PROGRAM MAIN
VAR
	fbGetCurTaskIdx  : GETCURTASKINDEX;
	
	Layout : Buffer_Layout;
	Buffer : ARRAY[0..63] OF BYTE;
	
	// out var
	VarEen : INT;
	VarTwee : INT;
END_VAR


Set_Buffer_Layout(
	Buffer_Size:= 64, 
	Bool_Amount:= 0, 
	Int_Amount:= 0, 
	Real_Amount:= 0, 
	String_Amount:= 2, 
	Layout:= Layout);

Set_Int_From_Buffer(
	In:= 300, 
	Num:= 0, 
	Layout:= Layout, 
	Buffer:= Buffer);
	
Set_Int_From_Buffer(
	In:= 30, 
	Num:= 1, 
	Layout:= Layout, 
	Buffer:= Buffer);
	
Set_Bool_Fom_Buffer(
	In:= TRUE, 
	Num:= 0, 
	Layout:= Layout, 
	Buffer:= Buffer);
	
	
Set_Bool_Fom_Buffer(
	In:= TRUE, 
	Num:= 1, 
	Layout:= Layout, 
	Buffer:= Buffer);
	
	
Set_Real_From_Buffer(
	In:= 3.55, 
	Num:= 0, 
	Layout:= Layout, 
	Buffer:= Buffer);
	
Set_Real_From_Buffer(
	In:= 10.66, 
	Num:= 1, 
	Layout:= Layout, 
	Buffer:= Buffer);
	
	
Set_String_From_Buffer(
	In:= 'AAAAA', 
	Num:= 0, 
	Layout:= Layout, 
	Buffer:= Buffer);
	
Set_String_From_Buffer(
	In:= 'AAAAAAAA', 
	Num:= 1, 
	Layout:= Layout, 
	Buffer:= Buffer);

END_PROGRAM

(* stored: Version 1.1.0.1, ProductVersion 3.1.4024.10
   POU MAIN: Id {ac7ccafc-0f66-4244-bca1-474ce436e2ea}, SpecialFunc None *)
